FUNCTION_BLOCK FINAL FB_AnalogueInput EXTENDS FB_EventLogger
VAR_IN_OUT
	Control					: ST_System;
END_VAR
VAR
	_Input		AT %I*		: UINT;					//Raw Input 1 - Analogue
	_Input2		AT %I*		: BOOL;					//Raw Input 2 - Digital
	_InputLimitHigh			: REAL;					//HighHigh limit of Raw Input 1
	_InputLimitLow			: REAL;					//Low limit of Raw Input 1
	_InputLimitHighHigh		: REAL;					//HighHigh limit of Raw Input 1
	_InputLimitLowLow		: REAL;					//LowLow limit of Raw Input 1
	_ManOnQa				: BOOL;					//Manual On Analogue Input
	_ManQa					: REAL;					//Manual Analogue Input
	_ManOn					: BOOL;					//Manual On
	_ManOff					: BOOL;					//Manual Off
	_ForceOn				: BOOL;					//Force On
	_ForceOff				: BOOL;					//Force Off
	_Fault					: BOOL;					//Fault
	_SimInput				: BOOL;		        	//Simulates Analogue Input
	_SimInput2				: BOOL;					//Simulates Digital Input
	_SimInputQa				: REAL;					//Value of Simulated Analogue Input
	_Value_Q	AT %Q*		: BOOL;					//Value of Input - Digital
	_Value_Qa	AT %Q*		: REAL;					//Value of Input - Analogue
	_FallingEdge			: BOOL;					//Falling Edge of Value Signal
	_RisingEdge				: BOOL;					//Raising Edge of Value Signal
	_DebounceOn_ET			: REAL;					//Debounce On Elapsed Time
	_DebounceOff_ET			: REAL;					//Debounce Off Elapsed Time
	_FaultTimer_ET			: REAL;					//Fault timer elapsed
	_Alarm					: BOOL;					//Device Alarm
	_Warning				: BOOL;					//Device Warning
	_AlarmNum				: DINT;					//Device Alarm Number
	_WarningNum				: DINT;					//Device Warning Number
	_riseEdge				: R_TRIG;				//Rising Edge Value Trigger
	_fallEdge				: F_TRIG;				//Falling Edge Value Trigger
	_Scale_Max				: REAL;					//Current Maximum (mA)
	_Scale_Min				: REAL;					//Current minimum (mA)
	_Scale_Value			: REAL;					//Current Value (mA)
	_Bit_Value				: REAL;					//Analogue Value Input
	_Bit_Max				: REAL;					//Maximum Bit Value (typically 32767)
	_Bit_Min				: REAL;					//Minimum Bit Value (typically 0)
	_Physical_Min			: REAL;					//Minimum Physical Value
	_Physical_Max			: REAL;					//Maximum Physical Value
	_ConfInput				: BOOL;					//Confirgured Input
	_DebounceOn_DN			: BOOL;					//Debounce On Timer is Done
	_DebounceOff_DN			: BOOL;					//Debounce Off Timer is Done
	_R_Trig					: ARRAY[0..9] OF R_TRIG;//Private Rising Edge Triggers
END_VAR
VAR PERSISTENT
	_Name					: STRING[15];			//Name for HMI
	_Description			: STRING[40];			//Description for HMI
	_AlarmMute				: BOOL;					//Alarm Mute
	_TypeConfig				: E_AInputTypeConfig;	//Type congifuration
	_DebounceOn_PT			: REAL;					//Debounce on timer preset time
	_DebounceOff_PT			: REAL;					//Debounce off timer preset time
	_FaultTimer_PT			: REAL;					//Fault timer preset time
	_HighAlarmLimit			: BOOL;					//Input Value is approaching the maximum operating limit.
	_LowAlarmLimit			: BOOL;					//Input Value is approaching the minimum operating limit.
	_HighHighAlarmLimit		: BOOL;					//Input Value is above  the maximum operating limit
	_LowLowAlarmLimit		: BOOL;					//Input Value is below the minimum operating limit.
	_BitValue_Max			: INT;					//Maximum Bit Value (typically 32767)
	_BitValue_Min			: INT;					//Minimum Bit Value (typically 0)
	_PhysicalValue_Min		: INT;					//Minimum Physical Value
	_PhysicalValue_Max		: INT;					//Maximum Physical Value
	_ScaleValue_Min			: INT;					//Minimum Scale Value				
	_ScaleValue_Max			: INT;					//Maximum Scale Value
END_VAR

M_TypeConfig();
M_AlarmMonitor();
M_WarningMonitor();
M_UnlatchManuals();
M_Output();

//Debounce On Timer
IF _ConfInput = TRUE AND NOT _ForceOff AND NOT _ManOff THEN
	_DebounceOn_ET := _DebounceOn_ET + Control.SystemTime.ScanTime;
	_debounceOn_DN := _DebounceOn_ET > _DebounceOn_PT;
ELSE
	_debounceOn_DN := FALSE;
END_IF
IF _debounceOn_DN OR _ForceOn OR _ManOn THEN
	_Value_Q := TRUE;
	_DebounceOff_ET := 0;
END_IF

//Debounce Off Timer
IF _ConfInput = FALSE AND NOT _ForceOn AND NOT _ManOn THEN
	_DebounceOff_ET := _DebounceOff_ET + Control.SystemTime.ScanTime;
	_debounceOff_DN := _DebounceOff_ET > _DebounceOff_PT;
ELSE
	_debounceOff_DN := FALSE;
END_IF
IF _debounceOff_DN OR _ForceOff OR _ManOff THEN
	_Value_Q:= FALSE;
	_DebounceOn_ET := 0;
END_IF

//Rising Edge Trigger 
_riseEdge(CLK := _Value_Q);
_RisingEdge := _riseEdge.Q;

//Falling Edge Trigger
_fallEdge(CLK := _Value_Q);
_FallingEdge := _fallEdge.Q;

{attribute 'monitoring' := 'variable'}
PROPERTY PUBLIC Alarm : Bool
GET
Alarm := _Alarm;
END_GET
END_PROPERTY

{attribute 'monitoring' := 'variable'}
PROPERTY PUBLIC AlarmMute : BOOL
SET
AlarmMute := _AlarmMute;
END_SET
END_PROPERTY

{attribute 'monitoring' := 'variable'}
PROPERTY PUBLIC DebounceOff_ET : real
GET
DebounceOff_ET := _DebounceOff_ET;
END_GET
END_PROPERTY

{attribute 'monitoring' := 'variable'}
PROPERTY PUBLIC DebounceOff_PT : real
GET
DebounceOff_PT := _DebounceOff_PT;
END_GET
SET
_DebounceOff_PT := DebounceOff_PT;
END_SET
END_PROPERTY

{attribute 'monitoring' := 'variable'}
PROPERTY PUBLIC DebounceOn_ET : real
GET
DebounceOn_ET := _DebounceOn_ET;
END_GET
END_PROPERTY

{attribute 'monitoring' := 'variable'}
PROPERTY PUBLIC DebounceOn_PT : real
GET
DebounceOn_PT := _DebounceOn_PT;
END_GET
SET
_DebounceOn_PT := DebounceOn_PT;
END_SET
END_PROPERTY

{attribute 'monitoring' := 'variable'}
PROPERTY PUBLIC Description : String[40]
GET
Description := _Description;
END_GET
SET
_Description := Description;
END_SET
END_PROPERTY

{attribute 'monitoring' := 'variable'}
PROPERTY PUBLIC FallingEdge : Bool
GET
FallingEdge := _FallingEdge;
END_GET
END_PROPERTY

{attribute 'monitoring' := 'variable'}
PROPERTY PUBLIC Fault : Bool
SET
_Fault := Fault;
END_SET
END_PROPERTY

{attribute 'monitoring' := 'variable'}
PROPERTY PUBLIC FaultTimer_ET : real
GET
FaultTimer_ET := _FaultTimer_ET;
END_GET
END_PROPERTY

{attribute 'monitoring' := 'variable'}
PROPERTY PUBLIC FaultTimer_PT : real
GET
FaultTimer_PT := _FaultTimer_PT;
END_GET
SET
_FaultTimer_PT := FaultTimer_PT;
END_SET
END_PROPERTY

{attribute 'monitoring' := 'variable'}
PROPERTY PUBLIC ForceOn : Bool
GET
ForceOn := _ForceOn;
END_GET
SET
_ForceOn := ForceOn;
END_SET
END_PROPERTY

{attribute 'monitoring' := 'variable'}
PROPERTY PUBLIC Input : UINT
GET
Input := _Input;
END_GET
END_PROPERTY

{attribute 'monitoring' := 'variable'}
PROPERTY PUBLIC Input2 : Bool
GET
Input2 := _Input2;
END_GET
END_PROPERTY

METHOD PRIVATE M_AlarmMonitor
VAR_INPUT
END_VAR
VAR_INST
END_VAR
VAR_INST // added by the converter: edge detectors and wires of the graphical bodies
    _w1, _w2, _w3, _w4, _w5 : BOOL;
    _rt1 : R_TRIG;
END_VAR
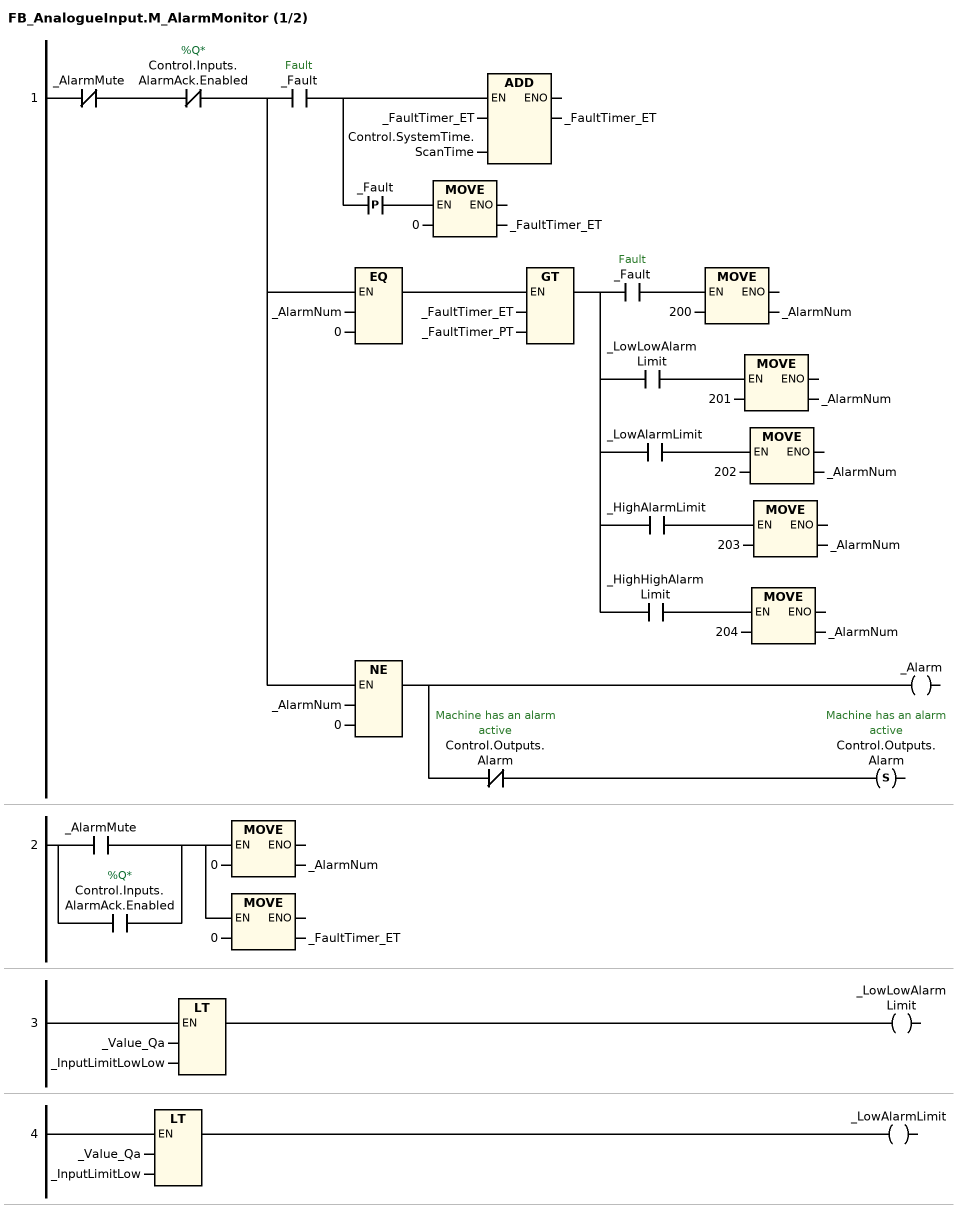
// NETWORK 1
//   Control.Inputs.AlarmAck.Enabled: AT %Q*
//   _Fault: Fault
//   _FaultTimer_ET: Fault timer elapsed
//   Control.SystemTime.ScanTime: Last scan time (Seconds)
//   _FaultTimer_PT: Fault timer preset time
//   Control.Outputs.Alarm: Machine has an alarm active
_w1 := NOT _AlarmMute AND NOT Control.Inputs.AlarmAck.Enabled;
_w2 := _w1 AND _Fault;
IF _w2 THEN _FaultTimer_ET := _FaultTimer_ET + Control.SystemTime.ScanTime; END_IF
_rt1(CLK := _Fault);
IF _w2 AND _rt1.Q THEN _FaultTimer_ET := 0; END_IF
_w3 := _w1 AND _AlarmNum = 0 AND _FaultTimer_ET > _FaultTimer_PT;
IF _w3 AND _Fault THEN _AlarmNum := 200; END_IF
IF _w3 AND _LowLowAlarmLimit THEN _AlarmNum := 201; END_IF
IF _w3 AND _LowAlarmLimit THEN _AlarmNum := 202; END_IF
IF _w3 AND _HighAlarmLimit THEN _AlarmNum := 203; END_IF
IF _w3 AND _HighHighAlarmLimit THEN _AlarmNum := 204; END_IF
_w4 := _w1 AND _AlarmNum <> 0;
_Alarm := _w4;
Control.Outputs.Alarm S= _w4 AND NOT Control.Outputs.Alarm;

// NETWORK 2
//   Control.Inputs.AlarmAck.Enabled: AT %Q*
//   _FaultTimer_ET: Fault timer elapsed
_w5 := _AlarmMute OR Control.Inputs.AlarmAck.Enabled;
IF _w5 THEN _AlarmNum := 0; END_IF
IF _w5 THEN _FaultTimer_ET := 0; END_IF

// NETWORK 3
_LowLowAlarmLimit := _Value_Qa < _InputLimitLowLow;

// NETWORK 4
_LowAlarmLimit := _Value_Qa < _InputLimitLow;

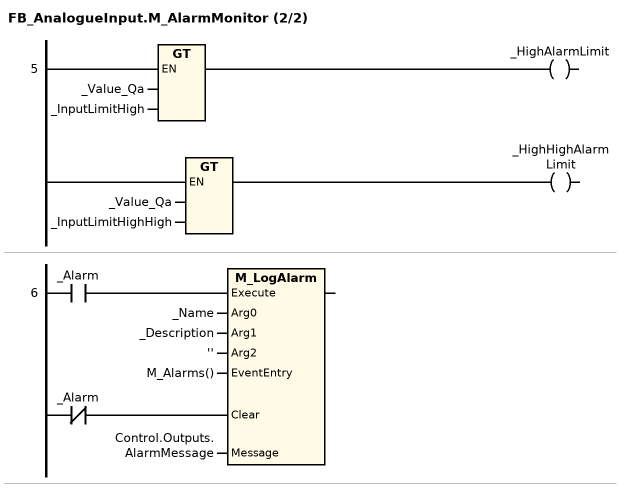
// NETWORK 5
_HighAlarmLimit := _Value_Qa > _InputLimitHigh;
_HighHighAlarmLimit := _Value_Qa > _InputLimitHighHigh;

// NETWORK 6
M_LogAlarm(Execute := _Alarm, Arg0 := _Name, Arg1 := _Description, Arg2 := '', EventEntry := M_Alarms(), Clear := NOT _Alarm, Message := Control.Outputs.AlarmMessage);
END_METHOD

METHOD PRIVATE M_Alarms : TcEventEntry
VAR_INPUT
END_VAR
CASE _AlarmNum OF
	201: M_Alarms:= TC_Events.TcAnalogueInput.A_201;//Low Low Limit Alarm
	202: M_Alarms:= TC_Events.TcAnalogueInput.A_202;//Low Limit Alarm			
	203: M_Alarms:= TC_Events.TcAnalogueInput.A_203;//High Limit Alarm
	204: M_Alarms:= TC_Events.TcAnalogueInput.A_204;//High High Limit Alarm							
ELSE
	M_Alarms:= TC_Events.TcAnalogueInput.A_Undefined;
END_CASE
END_METHOD

METHOD PRIVATE M_Output
VAR
END_VAR
VAR_INST
END_VAR
// Convert UINTs to INTs
_Scale_Min := ANY_TO_REAL(_ScaleValue_Min);
_Scale_Max := ANY_TO_REAL(_ScaleValue_Max);
_Bit_Value := ANY_TO_REAL(_Input);
_Bit_Max := ANY_TO_REAL(_BitValue_Max);		
_Bit_Min := ANY_TO_REAL(_BitValue_Min);		
_Physical_Min := ANY_TO_REAL(_PhysicalValue_Min);
_Physical_Max := ANY_TO_REAL(_PhysicalValue_Max);

IF _ManOnQa THEN
	_Value_Qa := _ManQa;
ELSIF _SimInput THEN
	_Value_Qa := _SimInputQa;
ELSIF _BitValue_Max <> 0 AND _PhysicalValue_Max <> 0 AND _ScaleValue_Max <> 0 THEN	
	// Calculate present electrical current value
	_Scale_Value := (((_Scale_Max - _Scale_Min)/F_CheckDivReal(divisor:=(_Bit_max - _Bit_min))) * (_Bit_Value - _Bit_min)) + _Scale_Min;

	// Convert electrical current value into measurable units
	_Value_Qa := (((_Physical_Max - _Physical_Min)/F_CheckDivReal(divisor:=(_Scale_Max - _Scale_Min))) * (_Scale_Value - _Scale_Min)) + _Physical_Min;	
END_IF
END_METHOD

METHOD PRIVATE M_TypeConfig
VAR_INPUT
END_VAR
VAR_INST
END_VAR
CASE _TypeConfig OF
	eAInputType_PLC_NO, eAInputType_SAFE_NO : 
		IF _Input2 OR _SimInput2 THEN
			_ConfInput := TRUE;
		ELSE
			_ConfInput := FALSE;
		END_IF
	eAInputType_PLC_NC, eAInputType_SAFE_NC : 
		IF NOT _Input2 OR _SimInput2 THEN
			_ConfInput := TRUE;
		ELSE
			_ConfInput := FALSE;
		END_IF
END_CASE
END_METHOD

METHOD PRIVATE M_UnlatchManuals
VAR_INPUT
END_VAR
VAR_INST
END_VAR
VAR_INST // added by the converter: edge detectors and wires of the graphical bodies
    _rt1, _rt2, _rt3 : R_TRIG;
END_VAR
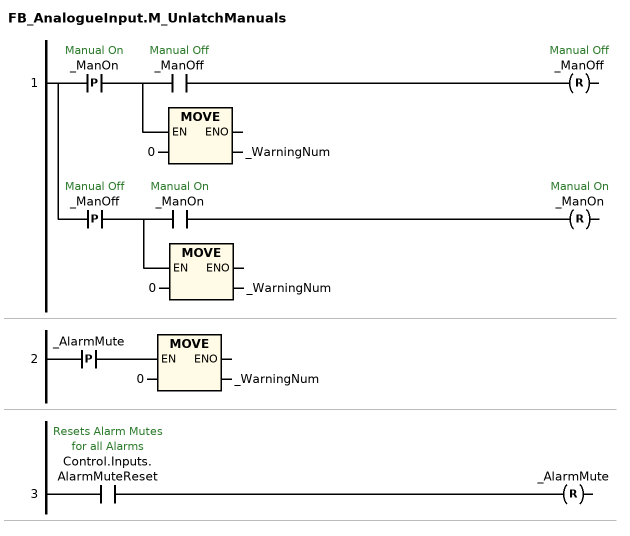
// NETWORK 1
//   _ManOn: Manual On
//   _ManOff: Manual Off
_rt1(CLK := _ManOn);
_ManOff R= _rt1.Q AND _ManOff;
IF _rt1.Q THEN _WarningNum := 0; END_IF
_rt2(CLK := _ManOff);
_ManOn R= _rt2.Q AND _ManOn;
IF _rt2.Q THEN _WarningNum := 0; END_IF

// NETWORK 2
_rt3(CLK := _AlarmMute);
IF _rt3.Q THEN _WarningNum := 0; END_IF

// NETWORK 3
//   Control.Inputs.AlarmMuteReset: Resets Alarm Mutes for all Alarms
_AlarmMute R= Control.Inputs.AlarmMuteReset;
END_METHOD

METHOD PRIVATE M_WarningMonitor
VAR_INPUT
END_VAR
VAR_INST
END_VAR
VAR_INST // added by the converter: edge detectors and wires of the graphical bodies
    _w1 : BOOL;
END_VAR
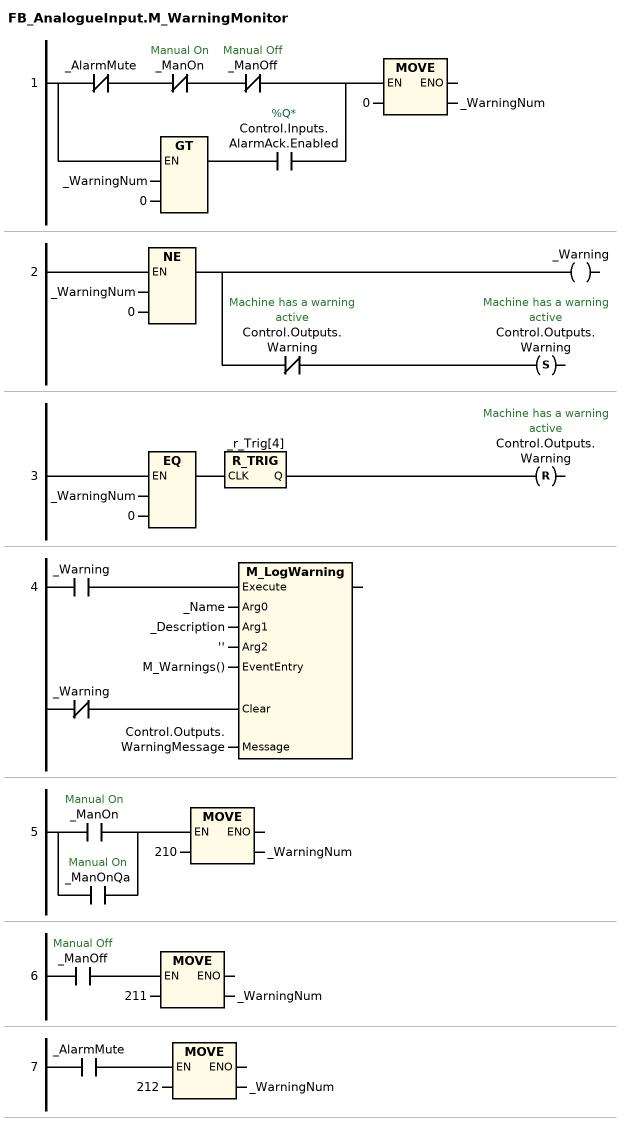
// NETWORK 1
//   _ManOn: Manual On
//   _ManOff: Manual Off
//   Control.Inputs.AlarmAck.Enabled: AT %Q*
IF NOT _AlarmMute AND NOT _ManOn AND NOT _ManOff OR _WarningNum > 0 AND Control.Inputs.AlarmAck.Enabled THEN
    _WarningNum := 0;
END_IF

// NETWORK 2
//   Control.Outputs.Warning: Machine has a warning active
_w1 := _WarningNum <> 0;
_Warning := _w1;
Control.Outputs.Warning S= _w1 AND NOT Control.Outputs.Warning;

// NETWORK 3
//   Control.Outputs.Warning: Machine has a warning active
_r_Trig[4](CLK := _WarningNum = 0); // R_TRIG
Control.Outputs.Warning R= _r_Trig[4].Q;

// NETWORK 4
M_LogWarning(Execute := _Warning, Arg0 := _Name, Arg1 := _Description, Arg2 := '', EventEntry := M_Warnings(), Clear := NOT _Warning, Message := Control.Outputs.WarningMessage);

// NETWORK 5
//   _ManOn: Manual On
//   _ManOnQa: Manual On
IF _ManOn OR _ManOnQa THEN _WarningNum := 210; END_IF

// NETWORK 6
//   _ManOff: Manual Off
IF _ManOff THEN _WarningNum := 211; END_IF

// NETWORK 7
IF _AlarmMute THEN _WarningNum := 212; END_IF
END_METHOD

METHOD PRIVATE M_Warnings : TcEventEntry
VAR_INPUT
END_VAR
CASE _WarningNum OF
	210: M_Warnings:= TC_Events.TcAnalogueInput.W_210;//Manual ON Enabled
	211: M_Warnings:= TC_Events.TcAnalogueInput.W_211;//Manual OFF Enabled			
	212: M_Warnings:= TC_Events.TcAnalogueInput.W_212;//Alarm Mute Active						
ELSE
	M_Warnings:=  TC_Events.TcAnalogueInput.W_Undefined;
END_CASE
END_METHOD

{attribute 'monitoring' := 'variable'}
PROPERTY PUBLIC ManOff : Bool
GET
ManOff := _ManOff;
END_GET
SET
_ManOff := ManOff;
END_SET
END_PROPERTY

{attribute 'monitoring' := 'variable'}
PROPERTY PUBLIC ManOn : Bool
GET
ManOn := _ManOn;
END_GET
SET
_ManOn := ManOn;
END_SET
END_PROPERTY

{attribute 'monitoring' := 'variable'}
PROPERTY PUBLIC ManOnQa : Bool
GET
ManOnQa := _ManOnQa;
END_GET
SET
_ManOnQa := ManOnQa;
END_SET
END_PROPERTY

{attribute 'monitoring' := 'variable'}
PROPERTY PUBLIC ManQa : REAL
GET
ManQa := _ManQa;
END_GET
SET
_ManQa := ManQa;
END_SET
END_PROPERTY

{attribute 'monitoring' := 'variable'}
PROPERTY PUBLIC Name : String[15]
GET
Name := _Name;
END_GET
SET
_Name := Name;
END_SET
END_PROPERTY

{attribute 'monitoring' := 'variable'}
PROPERTY PUBLIC RisingEdge : Bool
GET
RisingEdge := _RisingEdge;
END_GET
END_PROPERTY

{attribute 'monitoring' := 'variable'}
PROPERTY PUBLIC SimInput : Bool
SET
_SimInput := SimInput;
END_SET
END_PROPERTY

{attribute 'monitoring' := 'variable'}
PROPERTY PUBLIC SimInput2 : Bool
SET
_SimInput2 := SimInput2;
END_SET
END_PROPERTY

{attribute 'monitoring' := 'variable'}
PROPERTY PUBLIC SimInputQa : REAL
GET
SimInputQa := _SimInputQa;
END_GET
SET
_SimInputQa := SimInputQa;
END_SET
END_PROPERTY

{attribute 'monitoring' := 'variable'}
PROPERTY PUBLIC StandbyReset : Bool
GET
StandbyReset := _ForceOff;
END_GET
SET
_ForceOff := StandbyReset;
END_SET
END_PROPERTY

{attribute 'monitoring' := 'variable'}
PROPERTY PUBLIC Value_Q : BOOL
GET
Value_Q := _Value_Q;
END_GET
SET
_Value_Q := Value_Q;
END_SET
END_PROPERTY

{attribute 'monitoring' := 'variable'}
PROPERTY PUBLIC Value_Qa : REAL
GET
Value_Qa := _Value_Qa;
END_GET
SET
_Value_Qa := Value_Qa;
END_SET
END_PROPERTY

{attribute 'monitoring' := 'variable'}
PROPERTY PUBLIC Warning : Bool
GET
Warning := _Warning;
END_GET
END_PROPERTY

END_FUNCTION_BLOCK

(* stored: Version 1.1.0.1, ProductVersion 3.1.4024.3
   POU FB_AnalogueInput: Id {69e5f84c-e7bd-445b-8324-bd54e0fad752}, SpecialFunc None
   Property Alarm: Id {65212e95-ce1b-4c9e-b4b7-10fdfbfcf251}
   Get Get: Id {8e72e6c7-1cff-4a35-957e-ab9b8682b094}
   Property AlarmMute: Id {40051daa-3cda-459d-8795-0a03b156e922}
   Set Set: Id {8e58d88e-92ff-47c7-bf9c-45c8b5551c85}
   Property DebounceOff_ET: Id {8e008a3c-ae92-4d06-8817-7eb18e130ee6}
   Get Get: Id {69c2a982-a95d-4077-b6be-31ad2a8b863d}
   Property DebounceOff_PT: Id {769fc002-a9bb-4e4d-93ea-e188f771c610}
   Get Get: Id {64586291-91bc-4a9e-92de-cfe636673b02}
   Set Set: Id {d54ded2f-0dc1-40e4-81e1-3bd35ffeb738}
   Property DebounceOn_ET: Id {29d1cbc5-1db5-453a-b576-44ca1b38299d}
   Get Get: Id {5a19e36c-0879-44fa-a0bd-deca29eedac0}
   Property DebounceOn_PT: Id {c63b3a54-b5f9-4bb6-a6a5-1c2188dcf175}
   Get Get: Id {6cd4a671-0e2f-4fd5-87e6-1289b08aa17b}
   Set Set: Id {73f4fd73-b03a-463e-8df3-f97c70ffc781}
   Property Description: Id {94c4b75c-5ec4-4a97-a26f-ff0d8da1b530}
   Get Get: Id {469f79fd-7485-4e77-975d-f8f47acc36ae}
   Set Set: Id {7f475ff6-a75e-43a6-985e-ab6f4d63ab98}
   Property FallingEdge: Id {e78305d2-5d45-476a-8dd9-8e6f666d98c6}
   Get Get: Id {d387f643-38d7-4686-bf6a-2aeaefb7003e}
   Property Fault: Id {2e471ad8-a4e5-4313-8d7e-9de9a226e429}
   Set Set: Id {6282e5ca-015a-4a7c-a74c-0b40ea47aa91}
   Property FaultTimer_ET: Id {4dec0dcd-3ddd-4a11-8808-3cd2b8bfbf24}
   Get Get: Id {686953e6-71d9-4e24-91d0-aa0af9bab55b}
   Property FaultTimer_PT: Id {8b0b508e-d43b-44da-be42-e3fd1fa9760b}
   Get Get: Id {aaf41233-799c-476a-ab00-1f52912e25e7}
   Set Set: Id {278b1e3c-0829-4a39-9d9b-5ab94a3f35fc}
   Property ForceOn: Id {5f557302-c220-4297-8b45-a11ad5f63315}
   Get Get: Id {9763c847-d20f-4b9f-8a60-1f5cd4dc8d41}
   Set Set: Id {0cd48963-351d-46d5-ab3d-7fae191a485e}
   Property Input: Id {975acccc-9d26-49fb-a1c6-4153c1d179af}
   Get Get: Id {6779d31a-d41e-43e9-ae6d-e0571316cc60}
   Property Input2: Id {4c7c246c-fc31-4b62-8553-e167eaf7642d}
   Get Get: Id {3150179c-02e6-485e-b770-91dadc6e41f9}
   Method M_AlarmMonitor: Id {c34e5cae-4fab-4d6c-ab29-59839639fbab}
   Method M_Alarms: Id {7af2371c-fcd0-48a7-b955-d7aa8b81a5bd}
   Method M_Output: Id {a8f7c6a2-686c-44d2-8554-e4a516de40de}
   Method M_TypeConfig: Id {1e36ee77-39c2-4432-a557-51519cfe67d9}
   Method M_UnlatchManuals: Id {506219f8-9fa4-40a2-a1ef-f37cd235c47d}
   Method M_WarningMonitor: Id {85190806-04a9-4f3b-b633-be4e560259da}
   Method M_Warnings: Id {b560d1b3-9db0-44d1-be88-0ef4826bbfbf}
   Property ManOff: Id {6f94cc68-3d94-4e3b-9711-b067d69c7492}
   Get Get: Id {95b8f196-a991-4058-97b9-7335b91a1308}
   Set Set: Id {087c48ac-7f46-48c2-9913-8afee85292d8}
   Property ManOn: Id {33aedbb6-4b82-4872-b098-b0c7205a6c00}
   Get Get: Id {9fe70657-c8fe-4ac3-84a8-d3cc375ce5c2}
   Set Set: Id {90ebe990-f58c-4b31-b623-635dc28a0639}
   Property ManOnQa: Id {a6970a3d-9151-4cb1-83ab-0c3b18a27111}
   Get Get: Id {9c16c0d3-2740-4a72-8d6e-9688902053b6}
   Set Set: Id {31eee729-ef10-4eb0-b1e9-30103f892037}
   Property ManQa: Id {154fc6fa-32d5-4b9b-9179-9a90e472f4af}
   Get Get: Id {034630a5-0980-4251-98cf-a71d0378cfd9}
   Set Set: Id {8970ac90-70df-4db8-913a-cd9fdf829951}
   Property Name: Id {3626af5e-f3ea-4c3f-9f60-b69fe186b2fb}
   Get Get: Id {170bf006-36fc-4cd9-b751-f57c7e86c03a}
   Set Set: Id {196e83d5-8edf-4c12-bae9-f96730ec5bb8}
   Property RisingEdge: Id {31579b0a-89d2-4509-9bc1-663653f7e5bd}
   Get Get: Id {038fef2b-55fc-4896-ae24-f5a42729f27f}
   Property SimInput: Id {3c1fb3af-8d39-4ea2-b7c7-5b72312d168f}
   Set Set: Id {eefb275d-1b77-429c-a05f-c63111080604}
   Property SimInput2: Id {f8d05e2c-de8f-449c-a193-142d22e081c4}
   Set Set: Id {49ed9871-af14-472d-baef-d8653778bd47}
   Property SimInputQa: Id {69f72310-6599-4f1c-bc8c-faf51cc23cb2}
   Get Get: Id {8f5c92b7-46df-4f1e-8141-650d821d7889}
   Set Set: Id {e5349875-cdc9-4a50-a462-aaa3cdbefd5f}
   Property StandbyReset: Id {e38ecba7-c07e-4ff4-972c-c0ee0d499891}
   Get Get: Id {4a8b46f9-d37a-499d-bed7-0f0d56716a30}
   Set Set: Id {4f5bc544-2786-472c-b96c-009b94de046a}
   Property Value_Q: Id {abebdce7-2dfe-4298-bd0c-7fe48eafbe57}
   Get Get: Id {c8eee953-868b-4911-bd05-cfb1cbfc8a9e}
   Set Set: Id {cf5a771f-b775-47df-b827-d462b6108c94}
   Property Value_Qa: Id {cc2acfe3-4231-4038-bc15-72d391938fff}
   Get Get: Id {eb3617b7-832d-4e9b-91ba-2d79c1ff0bcf}
   Set Set: Id {7d429388-fa8f-4b42-b6f8-06a0466372f3}
   Property Warning: Id {6568cb09-a633-4d00-bd35-8b70a8e1c1a2}
   Get Get: Id {7b5e1084-f035-432d-8955-e33d1d422f3d} *)
